// TIA Portal V17 export
// export: Created 2025-04-11T04:54:23.9916689Z, ExportSetting WithDefaults, DisplayName Totally Integrated Automation Portal, DisplayVersion V17, DisplayName TIA Portal Openness, DisplayVersion V17, DisplayName TIA Portal Version Control Interface, DisplayVersion V17, DisplayName SINAMICS Startdrive Advanced, DisplayVersion V17, DisplayName SINAMICS Startdrive G130, G150, S120, S150, SINAMICS MV, S210, DisplayVersion V17, DisplayName SINAMICS Startdrive G110M, G120, G120C, G120D, G120P, G115D, DisplayVersion V17, DisplayName STEP 7 Professional, DisplayVersion V17, DisplayName STEP 7 Safety, DisplayVersion V17, DisplayName WinCC Advanced, DisplayVersion V17
TYPE "UDT_Device_HMI"
// stored: IsFailsafeCompliant false
   STRUCT
      IN_xManualStart : Bool;   // 手动启动
      IN_xManualStop : Bool;   // 手动停止
      OUT_uiState : UInt;   // 状态字(0=初始状态,1=已停止,2=已启动,3=正在启动,4=正在停止,5=停止故障,6=启动故障,7=设备报警)
   END_STRUCT;
END_TYPE
